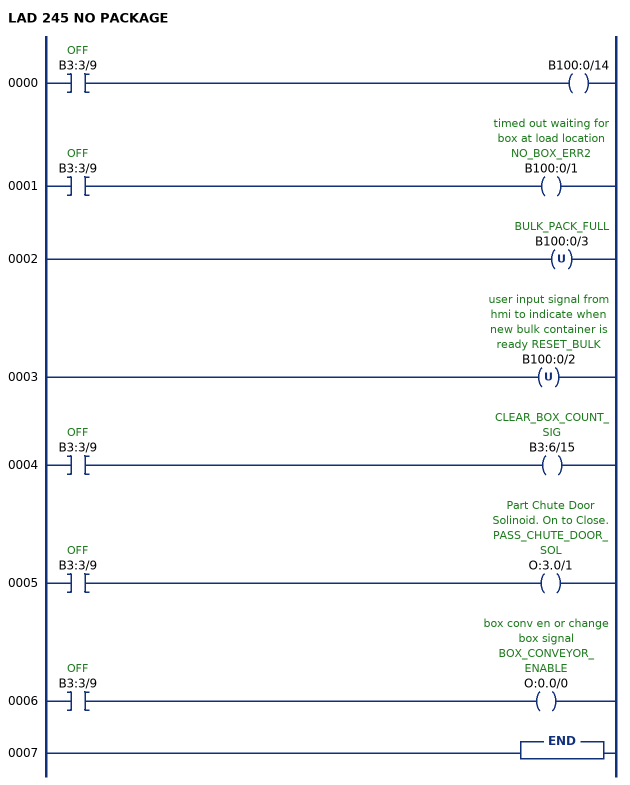
% Rung: 0 %
SOR XIC B3:3/9 OTE B100:0/14 EOR
%   B3:3/9  OFF %
% Rung: 1 %
SOR XIC B3:3/9 OTE B100:0/1 EOR
%   B3:3/9  OFF %
%   B100:0/1  NO_BOX_ERR2  "timed out waiting for box at load location" %
% Rung: 2 %
SOR OTU B100:0/3 EOR
%   B100:0/3  BULK_PACK_FULL %
% Rung: 3 %
SOR OTU B100:0/2 EOR
%   B100:0/2  RESET_BULK  "user input signal from hmi to indicate when new bulk container is ready" %
% Rung: 4 %
SOR XIC B3:3/9 OTE B3:6/15 EOR
%   B3:3/9  OFF %
%   B3:6/15  CLEAR_BOX_COUNT_SIG %
% Rung: 5 %
SOR XIC B3:3/9 OTE O:3.0/1 EOR
%   B3:3/9  OFF %
%   O:3.0/1  PASS_CHUTE_DOOR_SOL  "Part Chute Door Solinoid. On to Close." %
% Rung: 6 %
SOR XIC B3:3/9 OTE O:0.0/0 EOR
%   B3:3/9  OFF %
%   O:0.0/0  BOX_CONVEYOR_ENABLE  "box conv en or change box signal" %
% Rung: 7 %
SOR END EOR

LADDER 246 "RATE1"
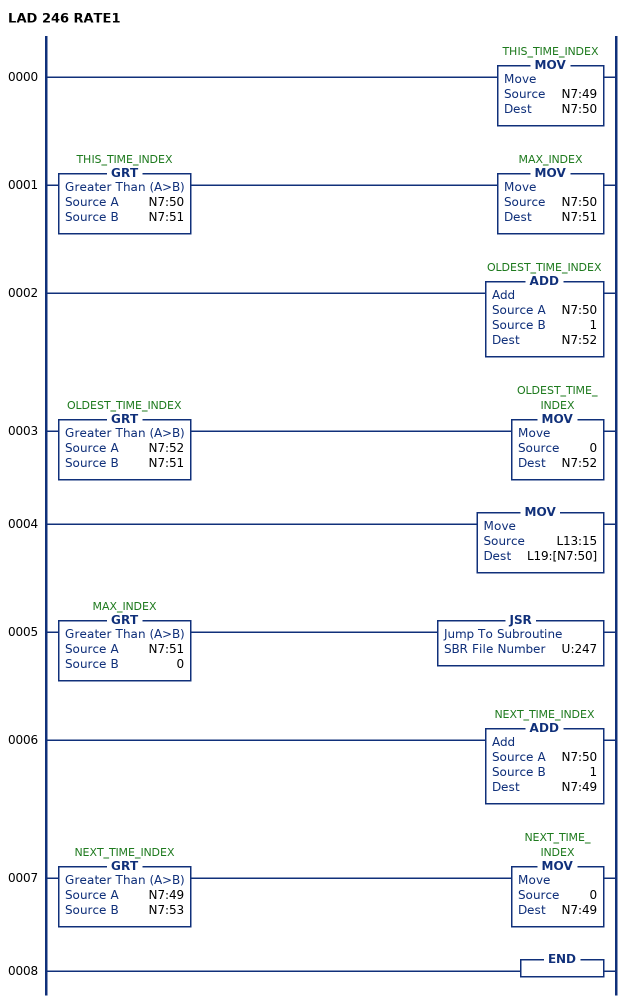
% Rung: 0 %
SOR MOV N7:49 N7:50 EOR
%   N7:49  NEXT_TIME_INDEX %
%   N7:50  THIS_TIME_INDEX %
% Rung: 1 %
SOR GRT N7:50 N7:51 MOV N7:50 N7:51 EOR
%   N7:50  THIS_TIME_INDEX %
%   N7:51  MAX_INDEX %
% Rung: 2 %
SOR ADD N7:50 1 N7:52 EOR
%   N7:50  THIS_TIME_INDEX %
%   N7:52  OLDEST_TIME_INDEX %
% Rung: 3 %
SOR GRT N7:52 N7:51 MOV 0 N7:52 EOR
%   N7:52  OLDEST_TIME_INDEX %
%   N7:51  MAX_INDEX %
% Rung: 4 %
SOR MOV L13:15 L19:[N7:50] EOR
%   L13:15  THE_TIME %
%   N7:50  THIS_TIME_INDEX %
% Rung: 5 %
SOR GRT N7:51 0 JSR U:247 EOR
%   N7:51  MAX_INDEX %
% Rung: 6 %
SOR ADD N7:50 1 N7:49 EOR
%   N7:50  THIS_TIME_INDEX %
%   N7:49  NEXT_TIME_INDEX %
% Rung: 7 %
SOR GRT N7:49 N7:53 MOV 0 N7:49 EOR
%   N7:49  NEXT_TIME_INDEX %
%   N7:53  UPPER_INDEX_LIMIT %
% Rung: 8 %
SOR END EOR

LADDER 247 "RATE2"
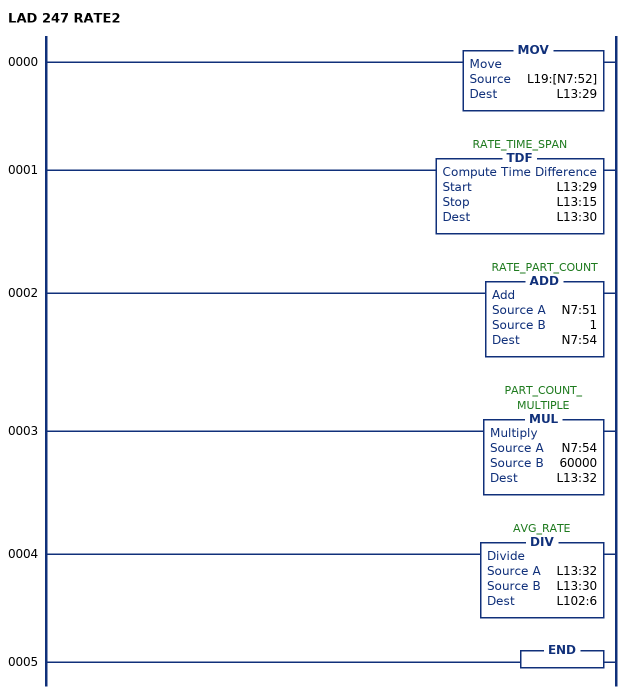
% Rung: 0 %
SOR MOV L19:[N7:52] L13:29 EOR
%   N7:52  OLDEST_TIME_INDEX %
% Rung: 1 %
SOR TDF L13:29 L13:15 L13:30 EOR
%   L13:15  THE_TIME %
%   L13:30  RATE_TIME_SPAN %
% Rung: 2 %
SOR ADD N7:51 1 N7:54 EOR
%   N7:51  MAX_INDEX %
%   N7:54  RATE_PART_COUNT %
% Rung: 3 %
SOR MUL N7:54 60000 L13:32 EOR
%   N7:54  RATE_PART_COUNT %
%   L13:32  PART_COUNT_MULTIPLE %
% Rung: 4 %
SOR DIV L13:32 L13:30 L102:6 EOR
%   L13:32  PART_COUNT_MULTIPLE %
%   L13:30  RATE_TIME_SPAN %
%   L102:6  AVG_RATE %
% Rung: 5 %
SOR END EOR

LADDER 248 "RESET RATE"
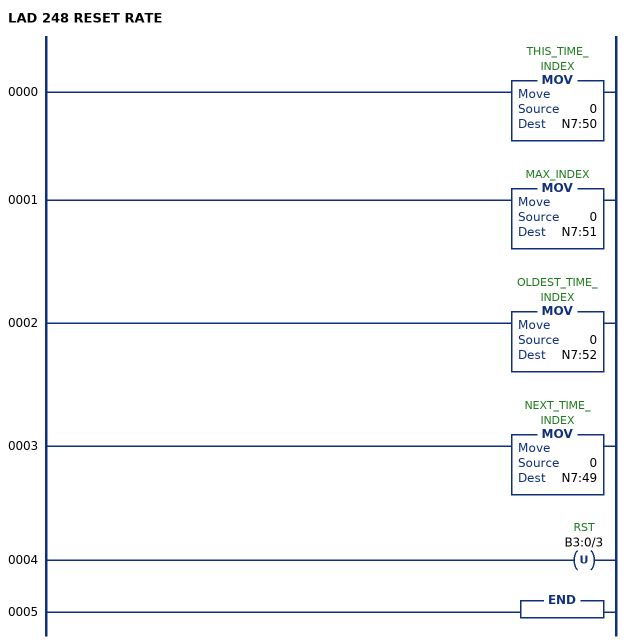
% Rung: 0 %
SOR MOV 0 N7:50 EOR
%   N7:50  THIS_TIME_INDEX %
% Rung: 1 %
SOR MOV 0 N7:51 EOR
%   N7:51  MAX_INDEX %
% Rung: 2 %
SOR MOV 0 N7:52 EOR
%   N7:52  OLDEST_TIME_INDEX %
% Rung: 3 %
SOR MOV 0 N7:49 EOR
%   N7:49  NEXT_TIME_INDEX %
% Rung: 4 %
SOR OTU B3:0/3 EOR
%   B3:0/3  RST %
% Rung: 5 %
SOR END EOR

LADDER 249 "NP STOP"    % stop on no good %
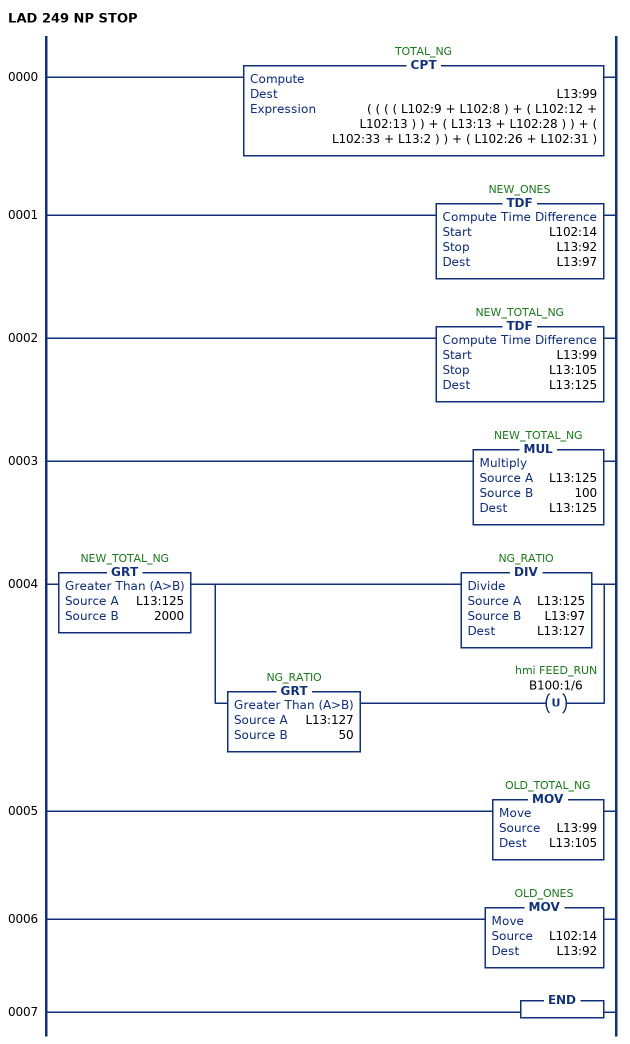
% Rung: 0 %
SOR CPT L13:99 " ( ( ( ( L102:9 + L102:8 ) + ( L102:12 + L102:13 ) ) + ( L13:13 + L102:28 ) ) + ( L102:33 + L13:2 ) ) + ( L102:26 + L102:31 ) " EOR
%   L13:99  TOTAL_NG %
%   L102:9  "too wide bottom" %
%   L102:8  "too close bottom" %
%   L102:12  "too close top count" %
%   L102:13  "too wide top count" %
%   L102:28  I1_I5_SKIPPEDCOUNT %
%   L102:33  I2_I6_SKIPPEDCOUNT %
%   L102:26  I1_I5_FAIL_COUNT %
%   L102:31  I2_I6_FAIL_COUNT %
% Rung: 1 %
SOR TDF L102:14 L13:92 L13:97 EOR
%   L102:14  ONES %
%   L13:92  OLD_ONES %
%   L13:97  NEW_ONES %
% Rung: 2 %
SOR TDF L13:99 L13:105 L13:125 EOR
%   L13:99  TOTAL_NG %
%   L13:105  OLD_TOTAL_NG %
%   L13:125  NEW_TOTAL_NG %
% Rung: 3 %
SOR MUL L13:125 100 L13:125 EOR
%   L13:125  NEW_TOTAL_NG %
% Rung: 4 %
SOR GRT L13:125 2000 BST DIV L13:125 L13:97 L13:127 NXB GRT L13:127 50 OTU B100:1/6 BND EOR
%   L13:125  NEW_TOTAL_NG %
%   L13:97  NEW_ONES %
%   L13:127  NG_RATIO %
%   B100:1/6  FEED_RUN  "hmi" %
% Rung: 5 %
SOR MOV L13:99 L13:105 EOR
%   L13:99  TOTAL_NG %
%   L13:105  OLD_TOTAL_NG %
% Rung: 6 %
SOR MOV L102:14 L13:92 EOR
%   L102:14  ONES %
%   L13:92  OLD_ONES %
% Rung: 7 %
SOR END EOR

LADDER 250 "SPEED BOT"    % high speed %
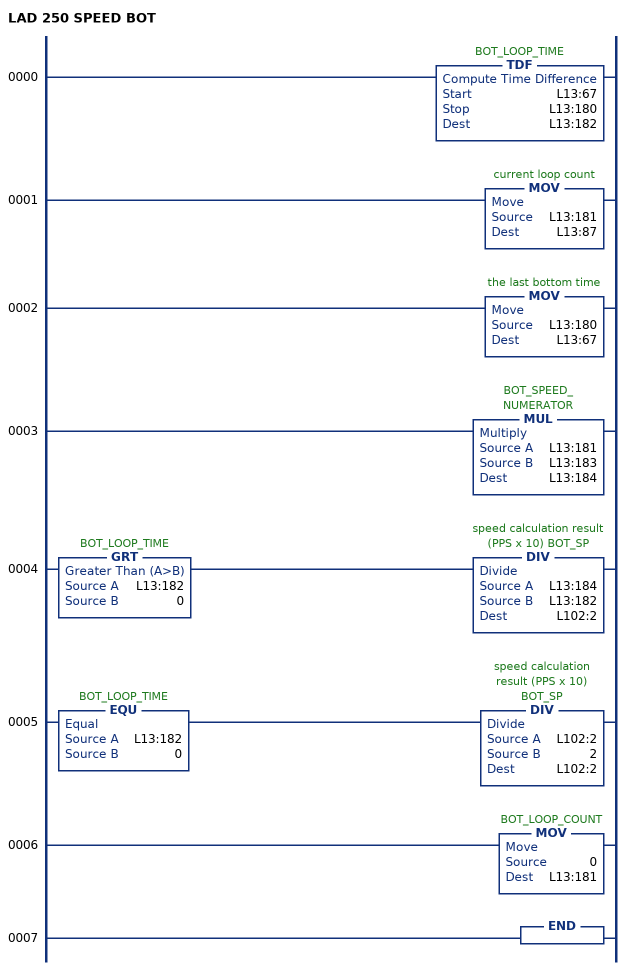
% Rung: 0 %
SOR TDF L13:67 L13:180 L13:182 EOR
%   L13:67  "the last bottom time" %
%   L13:180  BOT_THIS_TIME  "rtc bot belt movement event time" %
%   L13:182  BOT_LOOP_TIME %
% Rung: 1 %
SOR MOV L13:181 L13:87 EOR
%   L13:181  BOT_LOOP_COUNT %
%   L13:87  "current loop count" %
% Rung: 2 %
SOR MOV L13:180 L13:67 EOR
%   L13:180  BOT_THIS_TIME  "rtc bot belt movement event time" %
%   L13:67  "the last bottom time" %
% Rung: 3 %
SOR MUL L13:181 L13:183 L13:184 EOR
%   L13:181  BOT_LOOP_COUNT %
%   L13:183  TKS_PER_SECOND %
%   L13:184  BOT_SPEED_NUMERATOR %
% Rung: 4 %
SOR GRT L13:182 0 DIV L13:184 L13:182 L102:2 EOR
%   L13:182  BOT_LOOP_TIME %
%   L13:184  BOT_SPEED_NUMERATOR %
%   L102:2  BOT_SP  "speed calculation result (PPS x 10)" %
% Rung: 5 %
SOR EQU L13:182 0 DIV L102:2 2 L102:2 EOR
%   L13:182  BOT_LOOP_TIME %
%   L102:2  BOT_SP  "speed calculation result (PPS x 10)" %
% Rung: 6 %
SOR MOV 0 L13:181 EOR
%   L13:181  BOT_LOOP_COUNT %
% Rung: 7 %
SOR END EOR

LADDER 251 "SPEED TOP"    % high speed %
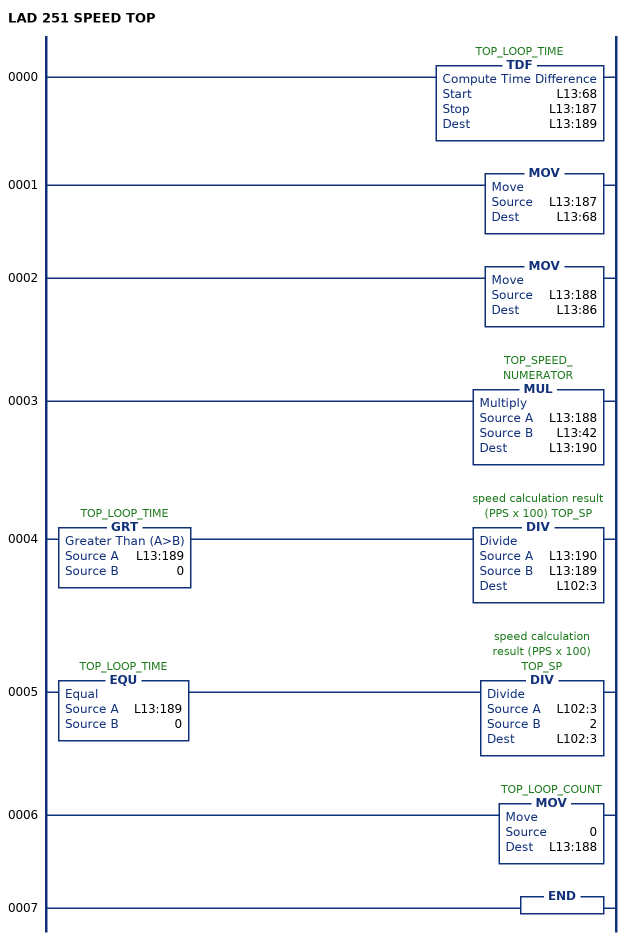
% Rung: 0 %
SOR TDF L13:68 L13:187 L13:189 EOR
%   L13:187  TOP_THIS_TIME  "rtc top belt movement event time" %
%   L13:189  TOP_LOOP_TIME %
% Rung: 1 %
SOR MOV L13:187 L13:68 EOR
%   L13:187  TOP_THIS_TIME  "rtc top belt movement event time" %
% Rung: 2 %
SOR MOV L13:188 L13:86 EOR
%   L13:188  TOP_LOOP_COUNT %
% Rung: 3 %
SOR MUL L13:188 L13:42 L13:190 EOR
%   L13:188  TOP_LOOP_COUNT %
%   L13:190  TOP_SPEED_NUMERATOR %
% Rung: 4 %
SOR GRT L13:189 0 DIV L13:190 L13:189 L102:3 EOR
%   L13:189  TOP_LOOP_TIME %
%   L13:190  TOP_SPEED_NUMERATOR %
%   L102:3  TOP_SP  "speed calculation result (PPS x 100)" %
% Rung: 5 %
SOR EQU L13:189 0 DIV L102:3 2 L102:3 EOR
%   L13:189  TOP_LOOP_TIME %
%   L102:3  TOP_SP  "speed calculation result (PPS x 100)" %
% Rung: 6 %
SOR MOV 0 L13:188 EOR
%   L13:188  TOP_LOOP_COUNT %
% Rung: 7 %
SOR END EOR

LADDER 252 "P BOT"    % high speed %
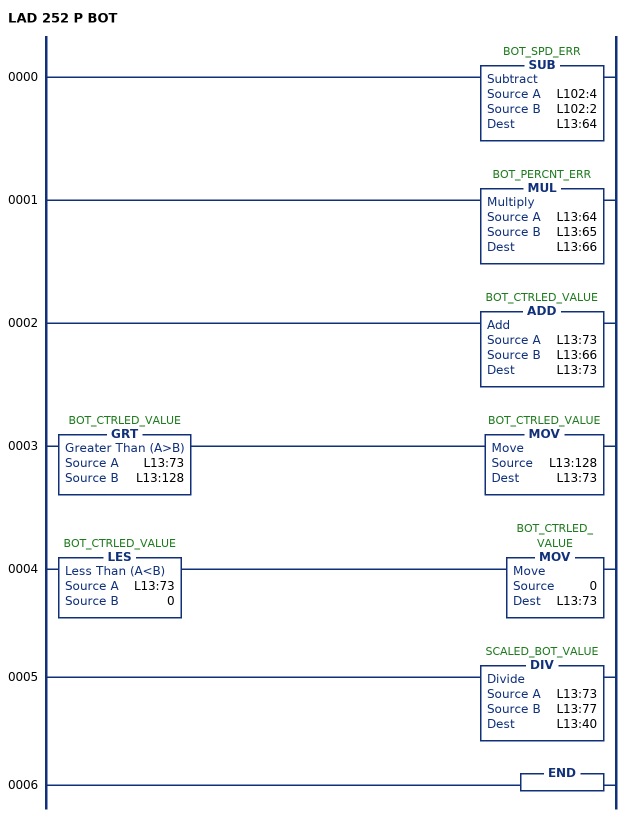
% Rung: 0 %
SOR SUB L102:4 L102:2 L13:64 EOR
%   L102:4  BOT_SPD_SETPOINT %
%   L102:2  BOT_SP  "speed calculation result (PPS x 10)" %
%   L13:64  BOT_SPD_ERR %
% Rung: 1 %
SOR MUL L13:64 L13:65 L13:66 EOR
%   L13:64  BOT_SPD_ERR %
%   L13:65  POS5SHIFT %
%   L13:66  BOT_PERCNT_ERR %
% Rung: 2 %
SOR ADD L13:73 L13:66 L13:73 EOR
%   L13:73  BOT_CTRLED_VALUE %
%   L13:66  BOT_PERCNT_ERR %
% Rung: 3 %
SOR GRT L13:73 L13:128 MOV L13:128 L13:73 EOR
%   L13:73  BOT_CTRLED_VALUE %
%   L13:128  "how much top has shifted since measurment" %
% Rung: 4 %
SOR LES L13:73 0 MOV 0 L13:73 EOR
%   L13:73  BOT_CTRLED_VALUE %
% Rung: 5 %
SOR DIV L13:73 L13:77 L13:40 EOR
%   L13:73  BOT_CTRLED_VALUE %
%   L13:40  SCALED_BOT_VALUE %
% Rung: 6 %
SOR END EOR

LADDER 253 "P TOP"    % high speed %
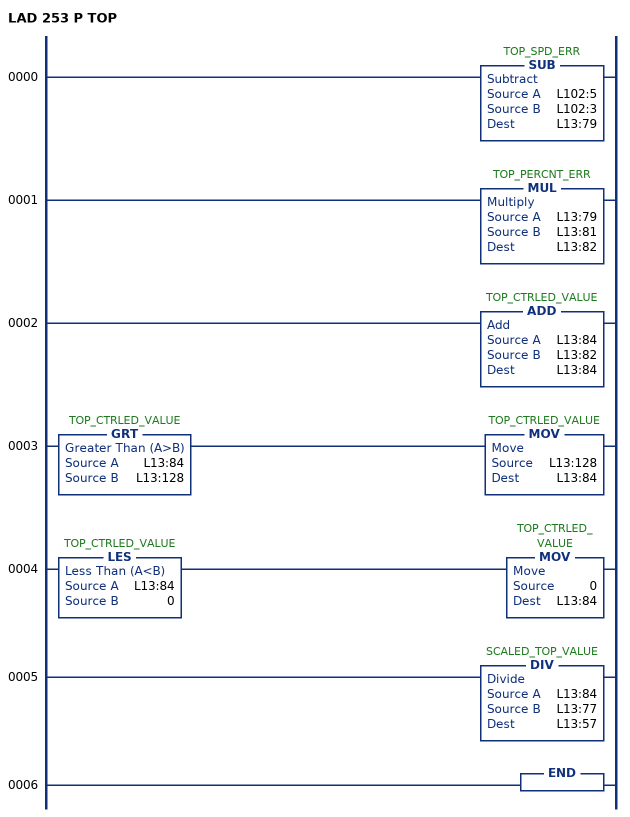
% Rung: 0 %
SOR SUB L102:5 L102:3 L13:79 EOR
%   L102:5  TOP_SPD_SETPOINT %
%   L102:3  TOP_SP  "speed calculation result (PPS x 100)" %
%   L13:79  TOP_SPD_ERR %
% Rung: 1 %
SOR MUL L13:79 L13:81 L13:82 EOR
%   L13:79  TOP_SPD_ERR %
%   L13:81  TOP_FDBK_RATIO %
%   L13:82  TOP_PERCNT_ERR %
% Rung: 2 %
SOR ADD L13:84 L13:82 L13:84 EOR
%   L13:84  TOP_CTRLED_VALUE %
%   L13:82  TOP_PERCNT_ERR %
% Rung: 3 %
SOR GRT L13:84 L13:128 MOV L13:128 L13:84 EOR
%   L13:84  TOP_CTRLED_VALUE %
%   L13:128  "how much top has shifted since measurment" %
% Rung: 4 %
SOR LES L13:84 0 MOV 0 L13:84 EOR
%   L13:84  TOP_CTRLED_VALUE %
% Rung: 5 %
SOR DIV L13:84 L13:77 L13:57 EOR
%   L13:84  TOP_CTRLED_VALUE %
%   L13:57  SCALED_TOP_VALUE %
% Rung: 6 %
SOR END EOR

LADDER 254 "TOTALCOUNT"
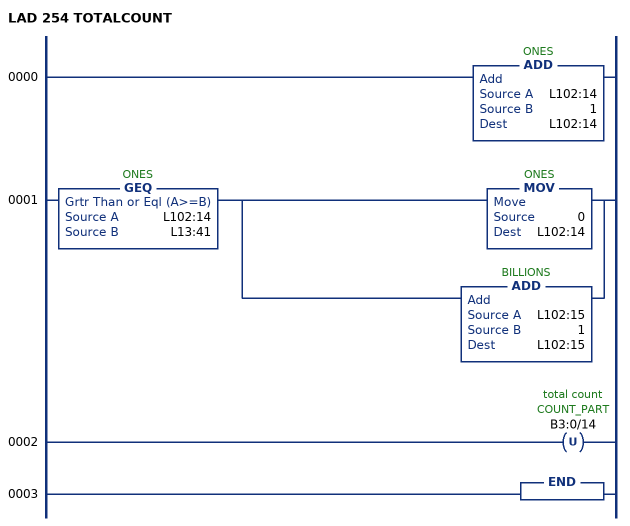
% Rung: 0 %
SOR ADD L102:14 1 L102:14 EOR
%   L102:14  ONES %
% Rung: 1 %
SOR GEQ L102:14 L13:41 BST MOV 0 L102:14 NXB ADD L102:15 1 L102:15 BND EOR
%   L102:14  ONES %
%   L13:41  "skipped count change in the last 3 seconds" %
%   L102:15  BILLIONS %
% Rung: 2 %
SOR OTU B3:0/14 EOR
%   B3:0/14  COUNT_PART  "total count" %
% Rung: 3 %
SOR END EOR

LADDER 255 "SAVED"
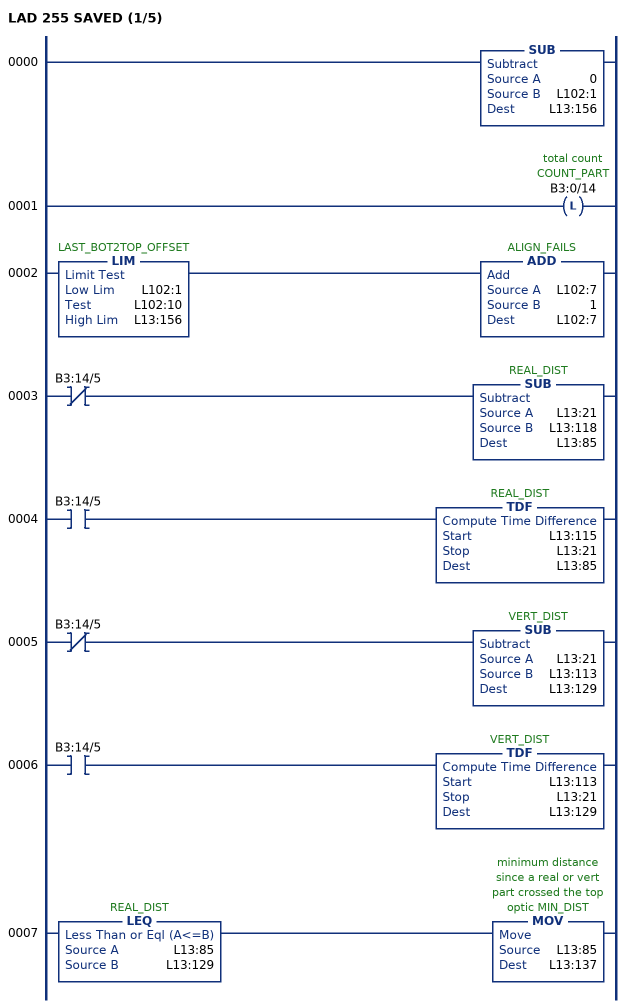
% Rung: 0 %
SOR SUB 0 L102:1 L13:156 EOR
%   L102:1  MAX_OFFSET  "transition zone width" %
% Rung: 1 %
SOR OTL B3:0/14 EOR
%   B3:0/14  COUNT_PART  "total count" %
% Rung: 2 %
SOR LIM L102:1 L102:10 L13:156 ADD L102:7 1 L102:7 EOR
%   L102:1  MAX_OFFSET  "transition zone width" %
%   L102:10  LAST_BOT2TOP_OFFSET %
%   L102:7  ALIGN_FAILS %
% Rung: 3 %
SOR XIO B3:14/5 SUB L13:21 L13:118 L13:85 EOR
%   L13:21  TOP_POSITION %
%   L13:118  REAL_CL_POSITION  "real part center line in raw position" %
%   L13:85  REAL_DIST %
% Rung: 4 %
SOR XIC B3:14/5 TDF L13:115 L13:21 L13:85 EOR
%   L13:115  TRAILING_EDGE_POS  "top optic trailing edge position" %
%   L13:21  TOP_POSITION %
%   L13:85  REAL_DIST %
% Rung: 5 %
SOR XIO B3:14/5 SUB L13:21 L13:113 L13:129 EOR
%   L13:21  TOP_POSITION %
%   L13:113  VIRT_CL_POSITION  "virtual part center line transfer from the bottom in raw position" %
%   L13:129  VERT_DIST %
% Rung: 6 %
SOR XIC B3:14/5 TDF L13:113 L13:21 L13:129 EOR
%   L13:113  VIRT_CL_POSITION  "virtual part center line transfer from the bottom in raw position" %
%   L13:21  TOP_POSITION %
%   L13:129  VERT_DIST %
% Rung: 7 %
SOR LEQ L13:85 L13:129 MOV L13:85 L13:137 EOR
%   L13:85  REAL_DIST %
%   L13:129  VERT_DIST %
%   L13:137  MIN_DIST  "minimum distance since a real or vert part crossed the top optic" %

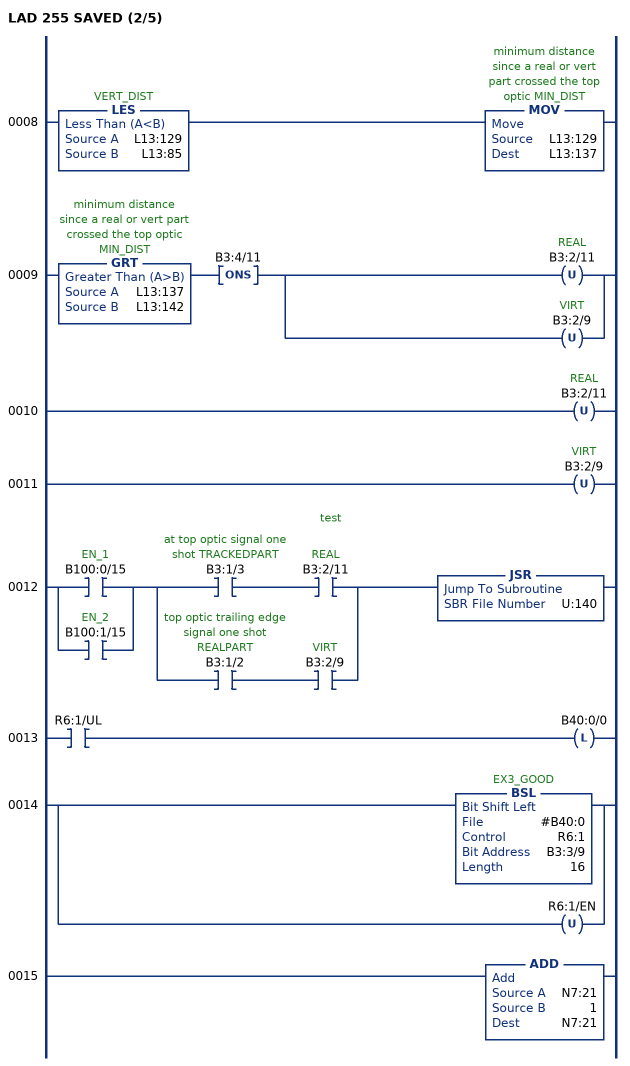
% Rung: 8 %
SOR LES L13:129 L13:85 MOV L13:129 L13:137 EOR
%   L13:129  VERT_DIST %
%   L13:85  REAL_DIST %
%   L13:137  MIN_DIST  "minimum distance since a real or vert part crossed the top optic" %
% Rung: 9 %
SOR GRT L13:137 L13:142 ONS B3:4/11 BST OTU B3:2/11 NXB OTU B3:2/9 BND EOR
%   L13:137  MIN_DIST  "minimum distance since a real or vert part crossed the top optic" %
%   L13:142  LAST_ALIGNMENT_FAILS %
%   B3:2/11  REAL %
%   B3:2/9  VIRT %
% Rung: 10 %
SOR OTU B3:2/11 EOR
%   B3:2/11  REAL %
% Rung: 11 %
SOR OTU B3:2/9 EOR
%   B3:2/9  VIRT %
% Rung: 12 %
% test %
SOR BST XIC B100:0/15 NXB XIC B100:1/15 BND BST XIC B3:1/3 XIC B3:2/11 NXB XIC B3:1/2 XIC B3:2/9 BND JSR U:140 EOR
%   B100:0/15  EN_1 %
%   B100:1/15  EN_2 %
%   B3:1/3  TRACKEDPART  "at top optic signal one shot" %
%   B3:2/11  REAL %
%   B3:1/2  REALPART  "top optic trailing edge signal one shot" %
%   B3:2/9  VIRT %
% Rung: 13 %
SOR XIC R6:1/UL OTL B40:0/0 EOR
% Rung: 14 %
SOR BST BSL #B40:0 R6:1 B3:3/9 16 NXB OTU R6:1/EN BND EOR
%   B40:0  EX3_GOOD %
%   B3:3/9  OFF %
% Rung: 15 %
SOR ADD N7:21 1 N7:21 EOR

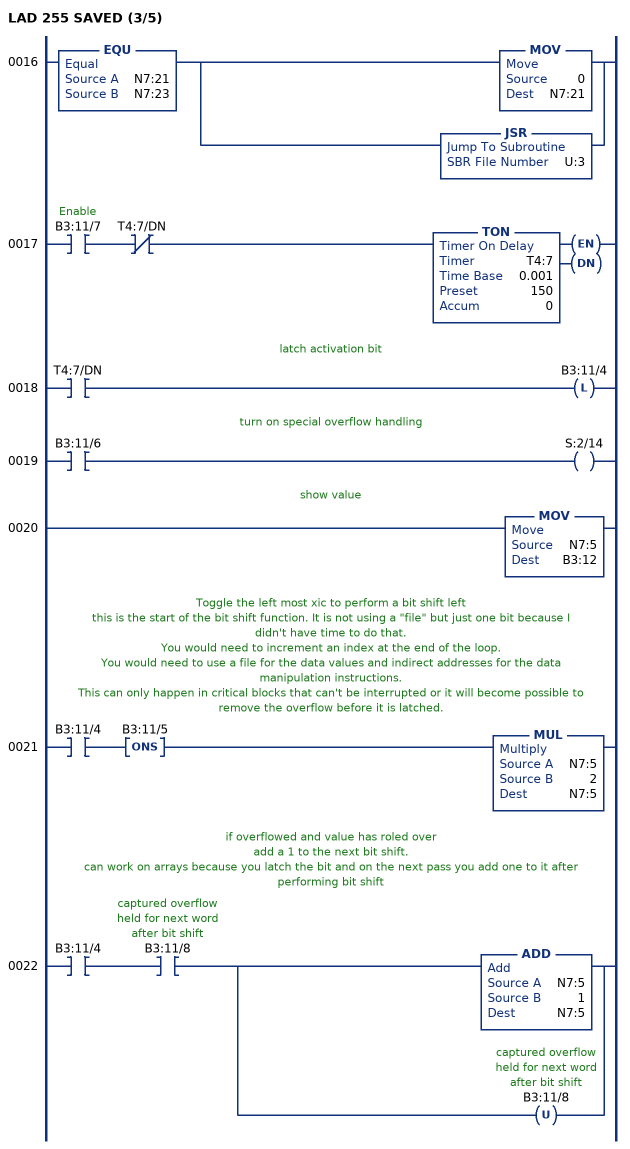
% Rung: 16 %
SOR EQU N7:21 N7:23 BST MOV 0 N7:21 NXB JSR U:3 BND EOR
% Rung: 17 %
SOR XIC B3:11/7 XIO T4:7/DN TON T4:7 0.001 150 0 EOR
%   B3:11/7  "Enable" %
% Rung: 18 %
% latch activation bit %
SOR XIC T4:7/DN OTL B3:11/4 EOR
% Rung: 19 %
% turn on special overflow handling %
SOR XIC B3:11/6 OTE S:2/14 EOR
% Rung: 20 %
% show value %
SOR MOV N7:5 B3:12 EOR
% Rung: 21 %
% Toggle the left most xic to perform a bit shift left
% 
% this is the start of the bit shift function. It is not using a "file" but just one bit because I didn't have time to do that.
% You would need to increment an index at the end of the loop.
% You would need to use a file for the data values and indirect addresses for the data manipulation instructions.
% 
% This can only happen in critical blocks that can't be interrupted or it will become possible to remove the overflow before it is latched. %
SOR XIC B3:11/4 ONS B3:11/5 MUL N7:5 2 N7:5 EOR
% Rung: 22 %
% if overflowed and value has roled over
% add a 1 to the next bit shift.
% can work on arrays because you latch the bit and on the next pass you add one to it after performing bit shift %
SOR XIC B3:11/4 XIC B3:11/8 BST ADD N7:5 1 N7:5 NXB OTU B3:11/8 BND EOR
%   B3:11/8  "captured overflow held for next word after bit shift" %

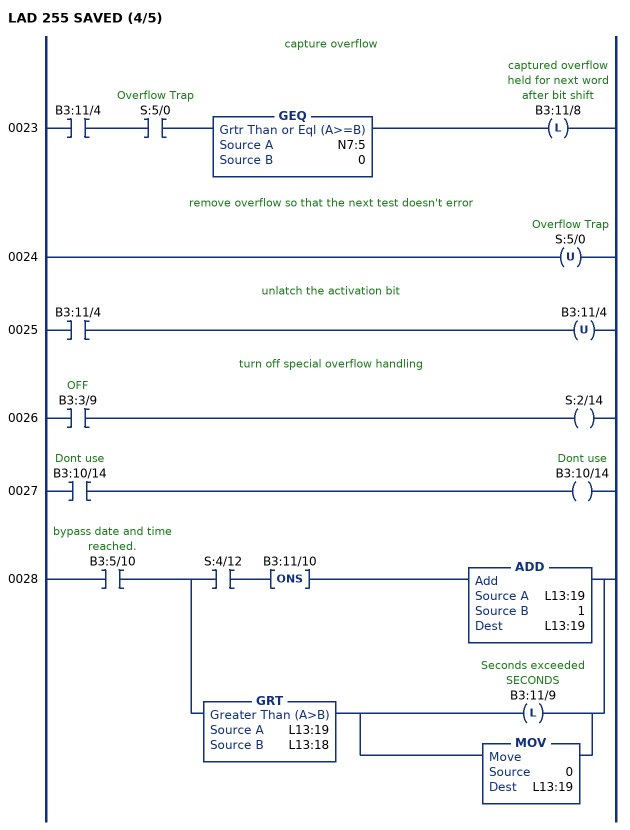
% Rung: 23 %
% capture overflow %
SOR XIC B3:11/4 XIC S:5/0 GEQ N7:5 0 OTL B3:11/8 EOR
%   S:5/0  "Overflow Trap" %
%   B3:11/8  "captured overflow held for next word after bit shift" %
% Rung: 24 %
% remove overflow so that the next test doesn't error %
SOR OTU S:5/0 EOR
%   S:5/0  "Overflow Trap" %
% Rung: 25 %
% unlatch the activation bit %
SOR XIC B3:11/4 OTU B3:11/4 EOR
% Rung: 26 %
% turn off special overflow handling %
SOR XIC B3:3/9 OTE S:2/14 EOR
%   B3:3/9  OFF %
% Rung: 27 %
SOR XIC B3:10/14 OTE B3:10/14 EOR
%   B3:10/14  "Dont use" %
% Rung: 28 %
SOR XIC B3:5/10 BST XIC S:4/12 ONS B3:11/10 ADD L13:19 1 L13:19 NXB GRT L13:19 L13:18 BST OTL B3:11/9 NXB MOV 0 L13:19 BND BND EOR
%   B3:5/10  "bypass date and time reached." %
%   L13:18  MAX %
%   B3:11/9  SECONDS  "Seconds exceeded" %

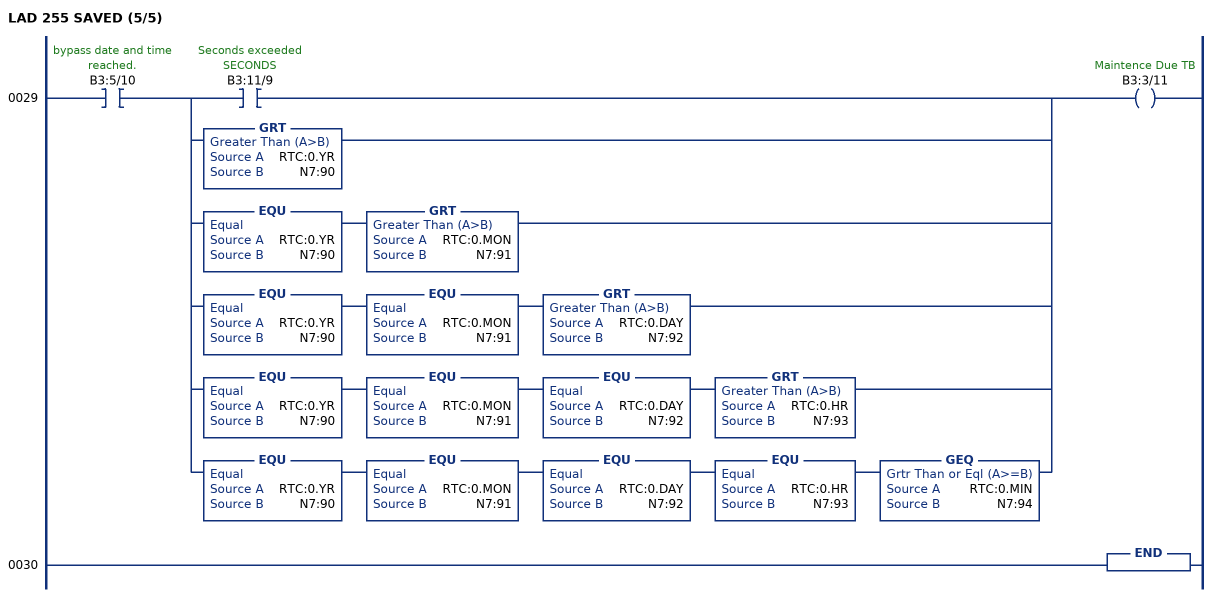
% Rung: 29 %
SOR XIC B3:5/10 BST XIC B3:11/9 NXB GRT RTC:0.YR N7:90 NXB EQU RTC:0.YR N7:90 GRT RTC:0.MON N7:91 NXB EQU RTC:0.YR N7:90 EQU RTC:0.MON N7:91 GRT RTC:0.DAY N7:92 NXB EQU RTC:0.YR N7:90 EQU RTC:0.MON N7:91 EQU RTC:0.DAY N7:92 GRT RTC:0.HR N7:93 NXB EQU RTC:0.YR N7:90 EQU RTC:0.MON N7:91 EQU RTC:0.DAY N7:92 EQU RTC:0.HR N7:93 GEQ RTC:0.MIN N7:94 BND OTE B3:3/11 EOR
%   B3:5/10  "bypass date and time reached." %
%   B3:11/9  SECONDS  "Seconds exceeded" %
%   N7:90  RTC %
%   B3:3/11  TB  "Maintence Due" %
% Rung: 30 %
SOR END EOR

OTHER DOCUMENTED ADDRESSES
  B38:0  EX1_GOOD
  B189:0/0  "change box"
  B189:0/9  "override boxing ok or not full signal"
  B189:0/11  "HMI force door close"
  B196:1/0  "Chute door is closed"
  B196:1/1  "control chute door"
  B196:1/13  "force box conveyor on"
  B196:3/0  "for hmi to continue production unlatched by hmi"
  HSC:0.0  "top"
  HSC:0.3/6  "Underflow interrupt"
  HSC:0.3/7  "Overflow interrupt"
  HSC:1.0  "bot"
  HSC:1.3/6  "Underflow interrupt"
  HSC:1.3/7  "Overflow interrupt"
  I7_TRAC  
  I:0.0/0  "Encoder Signal "A""
  I:0.0/1  "Encoder Signal "B""
  I:0.0/4  "Encoder Signal "A""
  I:0.0/5  "Encoder Signal "B""
  I:0.1/4  "not used"
  I:0.1/5  "not used"
  I:0.1/6  "not used"
  I:0.1/7  "not used"
  I:0.1/8  "not used"
  I:0.1/9  "not used"
  I:0.1/10  "not used"
  I:0.1/11  "not used"
  I:0.1/12  "not used"
  I:0.1/13  "not used"
  I:0.1/14  "not used"
  I:0.1/15  "not used"
  I:0.2  "not used"
  I:0.2/3  "Packaging Conveyor full"
  I:0.2/4  "Packaging Conveyor Box in Position"
  I:0.3  "not used"
  I:0.4  "Spare Analog Input 1"
  I:0.5  "Spare Analog Input 2"
  I:0.6  "Spare Analog Input 3"
  I:2.0/0  FRONT_ESTOP
  I:2.0/1  REAR_ESTOP
  I:2.0/8  FRONT_DOOR  "front door signal ce models only"
  I:2.0/9  REAR_DOOR  "rear door signal ce models only"
  I:2.0/11  "spare"
  L13:37  "loops"
  L13:132  "set speed"
  L13:133  "controlled speed"
  L23:19  TOP_OPT_FAIL_CT
  L23:34  AIR_PRESSURE_FAULT
  L28:0  INS_1_TIME
  L29:0  INS_1_POS
  L30:0  INS_5_TIME
  L31:0  INS_5_POS
  L32:0  INS_6_TIME
  L33:0  INS_6_POS
  L192:1  BOT_LAST_TIME  "rtc bot belt previous movement event time"
  L192:2  BOT_CYCLE_TIME  "rtc bot belt time between events"
  L192:7  FROM_REAL  "distance from real part signal at optic location"
  L192:8  FROM_TRACKED  "distance from tracked part signal at optic location"
  L192:16  TOP_LAST_TIME  "rtc top belt previous movement event time"
  L192:17  TOP_CYCLE_TIME  "rtc top belt time between events"
  L199:5  ACQTM51
  L199:6  ACQTM52
  L199:7  ACQTM53
  L199:9  "ones"
  L199:10  "billions"
  L199:13  DUMP_LONG
  L199:15  ACQTM11
  L199:16  ACQTM12
  L199:17  ACQTM13
  L199:20  RESULTTM1
  L199:22  CLEARTIME5COUNT
  L199:23  CLEARTIME6COUNT
  L199:24  ACQTM61
  L199:25  ACQTM62
  L199:26  ACQTM63
  L199:27  TMSINCETRIG1
  L199:29  TMSINCETRIG5
  L199:30  TMSINCETRIG6
  L199:31  CLEARTIME1COUNT
  L199:32  RESULTTM5
  L199:33  RESULTTM6
  L199:34  MAXACQTM1
  L199:36  MAXACQTM6
  N7  
  N101:2  I3_TRIG_LOC
  N101:3  I4_TRIG_LOC
  O:0.0/1  "spare"
  O:0.0/11  "Spare"
  O:0.0/12  "not used"
  O:0.0/13  "not used"
  O:0.0/14  "not used"
  O:0.0/15  "not used"
  O:0.1  "not used"
  O:0.2  "not used"
  O:0.3  "not used"
  O:0.5  "spare analog output"
  O:3.0/0  "spare"
  O:3.0/2  "spare"
  O:3.0/3  "light curtain range selection /* needed? */"
  O:3.0/7  "door unlocks on CE models"
  O:3.0/8  "Light?"
  O:3.0/9  NUT_HOPPER  "Nut Hopper Enable"
  O:3.0/11  NUT_FEEDER_AIR  "Nut Feeder Bowl Air Enable"
  PFILE:6  "check for part jams"
  PFILE:10  "Bottom belt HSC"
  PFILE:12  "Top belt HSC"
  Q2:55  END_OF_MAIN
  Q5:94  END_OF_BELTS
  T20:0  "Trigger On Time"
  U:9  "slow data"
  U:24  "check skipped fail rate"
  U:28  "faults"
  U:29  "speed"
  U:30  "count"
  U:31  "rate calc"
  U:32  "boxer"
  U:33  "bulk pack"
  U:34  "customer boxing unit signals"
  U:35  "cleanup"

COMMENTS NOT ATTACHED TO A CURRENT RUNG
  R6:2: B41 is the top good 3 file
  R6:11/DN: B39 is the top good 2 file
  R6:10/DN: B37 is the top good 1 file
  R6:6/DN: B35 is the top NG file
  R6:0: B36 is the bottom GOOD file
  R6:4: B34 is the bottom NG file
  R6:6: B35 is the top NG file
  R6:10: B37 is the top good 1 file

REVISION NOTES
  13: updated count reset
  14: added io moduals
  15: multiple steps toward new hmi integration
  21: test
  27: fix error if bulk pack and no boxing fallout were on

DATA TABLE (non-zero values as saved)
DATA B3
% B3:0 % 0X88A2 0X0160 0X4241 0X5101 0XE8B7 0X1540 0X0430 0X0061 0X5F80 0X2550
% B3:10 % 0X21E8 0X40C6 0X4000 0X1354 0X0001 0X0000 0X0000 0X0000 0X0000 0X0000
% B3:50 % 0X0001 0X0000 0X0000 0X0000 0X0000 0X0000 0X0000 0X0000 0X0000 0X0000
DATA T4
% .PRE .ACC %
% T4:0 % 0 3
% T4:1 % 150 0
% T4:2 % 400 0
% T4:3 % 222 95
% T4:4 % 1000 0
% T4:5 % 5 5
% T4:6 % 10 10
% T4:7 % 150 0
% T4:8 % 20 4
% T4:9 % 50 28
% T4:10 % 200 200
% T4:11 % 111 0
% T4:12 % 50 52
% T4:13 % 250 0
% T4:14 % 666 0
% T4:15 % 1000 1004
% T4:16 % 400 0
% T4:17 % 100 98
% T4:18 % 5 0
% T4:19 % 300 0
% T4:20 % 200 0
% T4:21 % 200 0
% T4:22 % 200 0
% T4:23 % 250 0
% T4:24 % 666 0
% T4:25 % 666 0
% T4:26 % 666 0
% T4:27 % 250 0
% T4:28 % 250 0
% T4:29 % 5000 0
% T4:30 % 333 0
% T4:31 % 444 353
% T4:32 % 222 91
% T4:33 % 222 91
% T4:34 % 1111 0
% T4:35 % 23 0
DATA C5
% .PRE .ACC %
% C5:0 % 32766 0
DATA R6
% .LEN .POS %
% R6:0 % 1250 0
% R6:1 % 16 0
% R6:2 % 1050 0
% R6:3 % 1050 0
% R6:4 % 1250 0
% R6:5 % 1250 0
% R6:6 % 1713 0
% R6:7 % 16 0
% R6:8 % 1024 0
% R6:9 % 3 0
% R6:10 % 1713 0
% R6:11 % 1050 0
% R6:12 % 10 0
% R6:13 % 10 0
% R6:14 % 10 0
% R6:15 % 10 0
% R6:16 % 1713 0
% R6:17 % 1713 0
% R6:18 % 1050 0
% R6:19 % 10 0
DATA N7
% N7:0 % 32767 3 870 128 3 0 0 0 500 43
% N7:10 % 1000 43 0 8 22 22 1000 2000 50 1050
% N7:20 % 0 1329 16 2000 0 48 0 0 0 250
% N7:30 % 666 32767 150 0 728 638 40 37 0 37
% N7:40 % 20 38 1 37 153 1218 705 1218 20 9
% N7:50 % 8 16 9 16 17 747 100 0 0 3
% N7:60 % 1713 1713 1050 868 1034 1024 4999 5 400 400
% N7:70 % 100 200 300 400 90 190 290 390 9931 32767
% N7:80 % 0 0 1269 1275 1278 1287 55 9 0 0
% N7:90 % 2011 4 4 12 1 55 9 222 222 12
% N7:100 % 1003 90 110 100 175 25 0 0 0 0
% N7:190 % -128 27477 27605 32767 0 0 0 0 0 0
DATA F8
% F8:0 % 6
DATA L13
% L13:0 % 210079 396779 0 226398 608693
% L13:5 % 0 168101 0 549882 132578
% L13:10 % 141024 4 0 15 90
% L13:15 % 1805434525 -2147483648 2147483647 2147483647 82058
% L13:20 % 504542469 -1157518992 777 0 100
% L13:25 % 49 0 -4598 0 1504741564
% L13:30 % 300692716 0 1020000 1551040931 1444
% L13:35 % 0 27 99 938346078 938346113
% L13:40 % 0 1000000000 1000000 1551040901 1550643757
% L13:45 % 1550643793 39 0 30 498757508
% L13:50 % 254790802 254393658 1504709068 0 0
% L13:55 % 254790766 254391598 4362 82392221 82397982
% L13:60 % 13239 1919711 0 600 -1
% L13:65 % 100 -100 -916487126 938337834 2
% L13:70 % 498758027 160 8 0 498757508
% L13:75 % 25 30 100 1551043121 2
% L13:80 % 557730 74 148 40 436232
% L13:85 % 274296 46 0 0 254790823
% L13:90 % 254790787 3 266458 5 1550643785
% L13:95 % 99 99608 0 1550643817 2320
% L13:100 % 7000 7 7200 1111 99610
% L13:105 % 2320 568360 498757383 25103 498757377
% L13:110 % 6 0 0 -1184299008 -1184401293
% L13:115 % -1184401287 6 3 -1184401290 1000
% L13:120 % 58 2994 27 121 469
% L13:125 % 0 498758027 2147483647 3276500 274297
% L13:130 % 9 18 0 249 -249
% L13:135 % 0 500 274296 1000 0
% L13:140 % 49 -49 36 50 50
% L13:145 % 254393734 5 254391674 5 9
% L13:150 % 12 20 102282 -102282 4
% L13:155 % 100 -10 0 37 4589052
% L13:160 % 6 28 24 1220 45
% L13:165 % -1184400897 -1184400888 -1184400897 -1184400888 6706
% L13:170 % 12817 11881 11881 800 200
% L13:175 % 4 4 42 23 38
% L13:180 % -916487126 0 0 1000000 0
% L13:185 % 0 0 938358909 19 51211
% L13:190 % 46000000 0 0 0 0
% L13:205 % 0 0 0 392968 411202
DATA L19
% L19:0 % 1550513632 1550547297 1550582696 1550591266 1550605120
% L19:5 % 1550613545 1550622393 1550630331 1550642212 1504741564
% L19:10 % 1504741989 1504744348 1504745725 1548569435 1550452362
% L19:15 % 1550456501 1550464224 0 0 0
DATA L20
% L20:0 % 1504718953 1504719464 1504719770 1504720366 1504720671
% L20:5 % 1504721119 1504723132 1504723532 1504723806 1504724893
% L20:10 % 1504725219 1504725560 1504726596 1504726913 1504727734
% L20:15 % 1504728008 1504729726 1504730599 1504742566 1504743110
% L20:20 % 1504743534 1504745890 1504747268 1548141170 1548141400
% L20:25 % 1548141630 1548141857 1548142087 1548142317 1548142548
% L20:30 % 1548142778 1548143008 1548143238 1548570979 1550346683
% L20:35 % 1550346914 1550347144 1550347373 1550347602 1550347831
% L20:40 % 1550348059 1550348288 1550348519 1550348746 1550453902
% L20:45 % 1550458041 1550465768 1550515177 1550548839 1550584242
% L20:50 % 1550592812 1550606665 1550615090 1550623940 1550631876
% L20:55 % 1550643757 1504697166 1504697440 1504697746 1504698044
% L20:60 % 1504698321 1504698603 1504698877 1504699155 1504699441
% L20:65 % 1504699718 1504700000 1504700298 1504700619 1504700900
% L20:70 % 1504701254 1504701543 1504701837 1504702158 1504702479
% L20:75 % 1504702825 1504703547 1504703833 1504704151 1504706976
% L20:80 % 1504707778 1504708711 1504708992 1504709270 1504709790
% L20:85 % 1504710302 1504712132 1504712413 1504712695 1504713159
% L20:90 % 1504713449 1504714226 1504714528 1504715187 1504715484
% L20:95 % 1504715762 1504716219 1504716965 1504717465 1504718045
DATA L21
% L21:0 % -1195974476 -1195974347 -1195974270 -1195974120 -1195974043
% L21:5 % -1195973930 -1195973423 -1195973322 -1195973253 -1195972979
% L21:10 % -1195972897 -1195972811 -1195972550 -1195972470 -1195972263
% L21:15 % -1195972194 -1195971761 -1195971541 -1195968525 -1195968388
% L21:20 % -1195968281 -1195967687 -1195967340 -1185031584 -1185031526
% L21:25 % -1185031468 -1185031410 -1185031352 -1185031294 -1185031236
% L21:30 % -1185031178 -1185031120 -1185031062 -1184923264 -1184475768
% L21:35 % -1184475710 -1184475652 -1184475595 -1184475537 -1184475479
% L21:40 % -1184475422 -1184475364 -1184475306 -1184475248 -1184448745
% L21:45 % -1184447702 -1184445754 -1184433302 -1184424817 -1184415897
% L21:50 % -1184413737 -1184410245 -1184408121 -1184405891 -1184403891
% L21:55 % -1184400897 -1195979966 -1195979897 -1195979820 -1195979745
% L21:60 % -1195979675 -1195979604 -1195979535 -1195979465 -1195979393
% L21:65 % -1195979323 -1195979252 -1195979177 -1195979096 -1195979025
% L21:70 % -1195978936 -1195978863 -1195978789 -1195978708 -1195978627
% L21:75 % -1195978540 -1195978358 -1195978286 -1195978206 -1195977494
% L21:80 % -1195977292 -1195977057 -1195976986 -1195976916 -1195976785
% L21:85 % -1195976656 -1195976195 -1195976124 -1195976053 -1195975936
% L21:90 % -1195975863 -1195975667 -1195975591 -1195975425 -1195975350
% L21:95 % -1195975280 -1195975165 -1195974977 -1195974851 -1195974705
DATA L22
% L22:0 % 1550465804 1550515213 1550548875 1550584278 1550592848
% L22:5 % 1550606701 1550615125 1550623976 1550631912 1550643793
% L22:10 % 1504723168 1504723568 1504723842 1504724929 1504725255
% L22:15 % 1504725596 1504726631 1504726948 1504727770 1504728044
% L22:20 % 1504729762 1504730635 1504742602 1504743146 1504743570
% L22:25 % 1504745926 1504747304 1548141217 1548141448 1548141677
% L22:30 % 1548141907 1548142137 1548142368 1548142598 1548142828
% L22:35 % 1548143058 1548143287 1548571015 1550346728 1550346955
% L22:40 % 1550347183 1550347414 1550347644 1550347873 1550348103
% L22:45 % 1550348333 1550348562 1550348793 1550453938 1550458077
DATA L23
% L23:0 % -1184445745 -1184433293 -1184424808 -1184415888 -1184413728
% L23:5 % -1184410236 -1184408112 -1184405882 -1184403882 -1184400888
% L23:10 % -1195973414 -1195973313 -1195973244 -1195972970 -1195972888
% L23:15 % -1195972802 -1195972541 -1195972461 -1195972254 -1195972185
% L23:20 % -1195971752 -1195971532 -1195968516 -1195968379 -1195968272
% L23:25 % -1195967678 -1195967331 -1185031572 -1185031514 -1185031456
% L23:30 % -1185031398 -1185031340 -1185031282 -1185031224 -1185031166
% L23:35 % -1185031108 -1185031050 -1184923255 -1184475757 -1184475700
% L23:40 % -1184475642 -1184475584 -1184475526 -1184475468 -1184475410
% L23:45 % -1184475353 -1184475295 -1184475237 -1184448736 -1184447693
DATA L30
% L30:0 % 1548142225 1548142453 1548142683 1548142912 1548143142
% L30:5 % 1548284776 1548562228 1550346587 1550346816 1550347045
% L30:10 % 1550347274 1550347503 1550347734 1550347963 1550348194
% L30:15 % 1550348424 1550348654 1550438038 1550440935 1550445151
% L30:20 % 1550449293 1550457018 1550506425 1550540086 1550575493
% L30:25 % 1550584060 1550597916 1550606340 1550615193 1550623122
% L30:30 % 1550635002 1550653925 1550693162 1550915373 1550927424
% L30:35 % 1550934775 1550941293 1551040901 1504720971 1504721846
% L30:40 % 1504733813 1504734356 1504734782 1504737144 1504738522
% L30:45 % 1548141073 1548141304 1548141532 1548141760 1548141991
DATA L31
% L31:0 % 498028993 498029051 498029109 498029166 498029224
% L31:5 % 498064918 498134841 498582526 498582583 498582641
% L31:10 % 498582699 498582757 498582815 498582873 498582931
% L31:15 % 498582989 498583047 498605571 498606301 498607364
% L31:20 % 498608407 498610354 498622808 498631291 498640215
% L31:25 % 498642374 498645865 498647989 498650220 498652218
% L31:30 % 498655212 498659980 498669868 498725873 498728910
% L31:35 % 498730763 498732405 498757508 487088307 487088527
% L31:40 % 487091543 487091680 487091787 487092382 487092729
% L31:45 % 498028703 498028761 498028818 498028876 498028934
DATA L32
% L32:0 % 1550442995 1550447211 1550451352 1550459077 1550508485
% L32:5 % 1550542145 1550577552 1550586120 1550599973 1550608400
% L32:10 % 1550617252 1550625181 1550637059 1550655984 1550695217
% L32:15 % 1550917435 1550929482 1550936834 1550943351 1551042961
% L32:20 % 1504709068 1504709522 1504710265 1504710767 1504711350
% L32:25 % 1504712261 1504712769 1504713075 1504713666 1504713976
% L32:30 % 1504714421 1504716438 1504716843 1504717113 1504718199
% L32:35 % 1504718525 1504718866 1504719901 1504720221 1504721035
% L32:40 % 1504721313 1504723031 1504723905 1504735875 1504736417
% L32:45 % 1504736842 1504739202 1504740577 1548141123 1548141575
DATA L33
% L33:0 % 498606820 498607883 498608926 498610873 498623327
% L33:5 % 498631810 498640734 498642893 498646384 498648508
% L33:10 % 498650739 498652737 498655731 498660499 498670387
% L33:15 % 498726392 498729429 498731282 498732924 498758027
% L33:20 % 487085307 487085422 487085609 487085735 487085882
% L33:25 % 487086112 487086240 487086317 487086466 487086544
% L33:30 % 487086656 487087164 487087266 487087334 487087608
% L33:35 % 487087690 487087776 487088037 487088118 487088323
% L33:40 % 487088393 487088826 487089046 487092062 487092199
% L33:45 % 487092306 487092901 487093248 498028715 498028829
DATA B35
% B35:110 % 0X0000 0X0000 0X0200 0X0000 0X0000 0X0000 0X0000 0X0000 0X0000 0X0000
DATA B37
% B37:0 % 0X0000 0X0000 0X2000 0X0000 0X0000 0X0000 0X0000 0X0000 0X0000 0X0000
DATA B40
% B40:0 % 0XAAAA
DATA B41
% B41:50 % 0X0000 0X0000 0X0000 0X0000 0X00C0 0X0000 0X0000 0X0000 0X0000 0X0000
DATA B100
% B100:0 % 0XA700 0X98A0 0X0004 0X0000 0X0000 0X0000 0X0000 0X0000 0X0000 0X0000
DATA N101
% N101:0 % 128 647 0 0 1182 111 867 1200 1200 1260
% N101:10 % 1269 1616 10 17693 491 0 3049 222 333 444
% N101:20 % 1000 500 400 0 0 0 222 222 0 0
DATA L102
% L102:0 % 50 10 1 901 0
% L102:5 % 900 0 13 0 0
% L102:10 % 4 11 0 0 266458
% L102:15 % 0 30 10 30 10
% L102:20 % 0 8 44 0 28
% L102:25 % 30 0 70 2295 0
% L102:30 % 160 10 72 0 0
% L102:35 % 0 9999999 0 999999 24
% L102:40 % 0 2 17124 0 0
